PROGRAM MAIN
VAR
END_VAR

END_PROGRAM

(* stored: Version 1.1.0.1
   POU MAIN: Id {c4180bb3-dc2f-44fa-beff-077cf1705622} *)
